RoboDK station: Basic HAMK Robotics station MG400.rdk

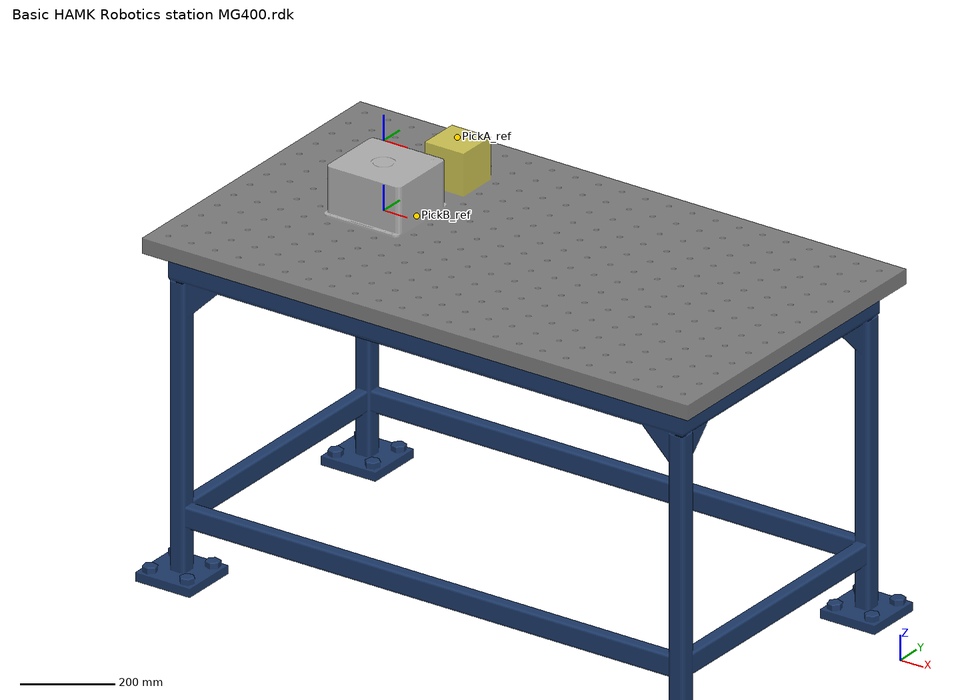
[picture v0: the station drawn from its stored meshes, robots at their saved joint values, targets as dots, program paths as lines]
Station HAMK Robotics Station MG400 (saved by RoboDK 5.6.7). Poses are relative to the parent item; angles as X-Y-Z fixed-axis rotations.
Station parameters (name, value as stored): LIN64
  - frame Dobot MG400 Base at (0, 0, 0) mm
    - robot Dobot MG400: 4 axes, payload 0.5 kg, reach 393.5 mm, repeatability 0.2 mm, weight 4 kg
        joint limits [-160, -25, -25, -360] to [160, 85, 105, 360]; home [0, 0, 0, 0]; saved at [-38.29, -5.611, 31.203, -38.3]
      - tool Suction Cup, TCP at (0, 0, 75.5) mm, size 42.6 x 40 x 76.8 mm
    - frame World at (0, 0, 0) mm
      - object Table 1400x800x800mm at (0, 0, 0) mm, size 1420 x 820 x 800 mm, geometry from Table-1400x800x800mm.sld
        - object HAMK logo at (360, 380, -115) mm, rotated rx 90 ry 0 rz 180 deg, size 301.4 x 100.9 x 9.4 mm, geometry from Fantastic Duup(2).stl
        - object white background at (360, 385.5, -110) mm, rotated rx 90 ry 0 rz 0 deg, size 480 x 184.8 x 2.4 mm, geometry from Fantastic Duup(3).stl
      - object box_ref at (50, 200, 50) mm, size 100 x 100 x 100 mm, geometry from box.sld
  - frame RefSuctionCup at (0, 0, 163) mm
    - target PickA_ref (Cartesian target) at (50, 200, -58) mm, rotated rx 180 ry 0 rz -179.99 deg; joints [75.964, 19.916, 77.779, 75.954] of Dobot MG400
    - target PickB_ref (Cartesian target) at (190, -150, -63) mm, rotated rx 180 ry 0 rz -179.99 deg; joints [-38.29, 27.304, 72.611, -38.3] of Dobot MG400
